KUKA KRL data list: FRAMELIB.dat

&ACCESS RV1
&REL 2
DEFDAT FRAMELIB PUBLIC

  STRUC VECTOR3DTYPE REAL X,Y,Z

  STRUC QUATERNIONTYPE REAL Q1,Q2,Q3,Q4

  STRUC AXISANGLETYPE REAL I,J,K,THETA

ENDDAT
